FUNCTION TryConvert_DATE_TO_LREAL : BOOL
VAR_INPUT
	in : DATE;
	out : REFERENCE TO LREAL;
END_VAR

out := DATE_TO_LREAL(in);
TryConvert_DATE_TO_LREAL := TRUE;

END_FUNCTION

(* stored: Version 1.1.0.1, ProductVersion 3.1.4024.12
   POU TryConvert_DATE_TO_LREAL: Id {849fbcce-b7e0-4214-8aa2-aad4a5c246c1}, SpecialFunc None *)
